// TIA Portal V17 export
// export: Created 2022-07-28T18:03:18.2436006Z, ExportSetting None, DisplayName Totally Integrated Automation Portal, DisplayVersion V17, DisplayName TIA Portal Openness, DisplayVersion V17, DisplayName TIA Portal Teamcenter Gateway, DisplayVersion V17, DisplayName TIA Portal Version Control Interface, DisplayVersion V17, DisplayName TIA Portal Test Suite Advanced, DisplayVersion V17, DisplayName SINAMICS Startdrive Advanced, DisplayVersion V17, DisplayName SINAMICS DCC, DisplayVersion V17, DisplayName SINAMICS Startdrive G130, G150, S120, S150, SINAMICS MV, S210, DisplayVersion V17, DisplayName SINAMICS Startdrive G110M, G120, G120C, G120D, G120P, G115D, DisplayVersion V17, DisplayName STEP 7 Professional, DisplayVersion V17, DisplayName SIMATIC Energy Suite, DisplayVersion V17, DisplayName STEP 7 CFC, DisplayVersion V17, DisplayName STEP 7 Safety, DisplayVersion V17, DisplayName WinCC Advanced / Unified PC, DisplayVersion V17, DisplayName SIMATIC Visualization Architect, DisplayVersion V17
TYPE "_ASensor_Config"
   STRUCT
      "b" { ExternalAccessible := 'False'; ExternalVisible := 'False'; ExternalWritable := 'False'} : Struct   // bool parameters
         AutoAskErrors { S7_SetPoint := 'True'} : Bool;
         AutoResetInterlock { S7_SetPoint := 'True'} : Bool;
         bit_2 { S7_SetPoint := 'True'} : Bool;
         bit_3 { S7_SetPoint := 'True'} : Bool;
         bit_4 { S7_SetPoint := 'True'} : Bool;
         bit_5 { S7_SetPoint := 'True'} : Bool;
         bit_6 { S7_SetPoint := 'True'} : Bool;
         bit_7 { S7_SetPoint := 'True'} : Bool;
      END_STRUCT;
      i_HMI_SensValRange { ExternalAccessible := 'False'; ExternalVisible := 'False'; ExternalWritable := 'False'} : Int;   // Range type of sensor val
      r_DisplayData { ExternalWritable := 'False'} : Real;   // Scaled data from senor (Output val)
      r_HH_Setpoint : Real := 90.0;   // Alarm Setpoint
      r_H_Setpoint : Real := 80.0;   // Warning Setpoint
      r_L_Setpoint : Real := 20.0;   // Warning Setpoint
      r_LL_Setpoint : Real := 10.0;   // Alarm Setpoint
      r_Hysteresis : Real := 2.0;   // High and low levels signals hysteresis
      r_WarnDetectTime : Real := 3.0;   // Delay for detecting alarms and warnings (filter), sec
      r_MaxVal : Real := 100.0;   // Max scaled sensor limit, eng unit
      r_MinVal : Real := 0.0;   // Min scaled sensor limit, eng unit
      r_MaxDisplayVal : Real := 100.0;   // Max scaled sensor displayed limit, eng unit
      r_MinDisplayVal : Real := 0.0;   // Min scaled sensor displayed limit, eng unit
      r_CurrMaxRange { ExternalWritable := 'False'} : Real := 100.0;   // Max range for current choiced display mode
      r_CurrMinRange { ExternalWritable := 'False'} : Real := 0.0;   // Min range for current choiced display mode
      r_Offset : Real := 0.0;   // Offset, eng unit
   END_STRUCT;
END_TYPE
